Omron Sysmac Studio project servo_limites (Sysmac Studio 1.23.0.14, StandardProject)

# Controller new_Controller_0: NX1P2-1040DT1 version 1.18
Axis eje_1, settings changed from default: AxisType=ServoType, UnitsConversion=EnumElement2, UnitsNumerator=8380608, UnitsDenominator=143, MaxVelocity=50, MaxJogVelocity=20, HomingMode=BackupAndPressingTime, StartDirection=NegativeDirection, OriginInputDetectionDirection=NegativeDirection, HomingVelocity=3, HomingApproachVelocity=1, HomingAcceleration=4, PushTime=1000, OriginCompensationValue=10, CompensationVelocity=0.5, ModuloMAXPosition=360, ModuloMINPosition=0, EncoderTypes=Abs
Task PrimaryTask (priority 4, period or condition 2000): Programa0

VAR_GLOBAL CONSTANT
    eje_1 : _sAXIS_REF;  (* at MC://_MC_AX[0] *)
END_VAR

PROGRAM Programa0
VAR
    servo_on : BOOL;
    et10 : BOOL;
    on_servo : BOOL;
    et11 : BOOL;
    et12 : BOOL;
    reset_servo1 : MC_Reset;
    power_servo1 : MC_Power;
    home_servo : MC_Home;
    absolute1_servo1 : MC_MoveAbsolute;
    abs_move : BOOL;
    et0 : BOOL;
    et1 : BOOL;
    et2 : BOOL;
    eje1 : _sAXIS_REF;
END_VAR
VAR_EXTERNAL CONSTANT
    eje_1 : _sAXIS_REF;
END_VAR

(* Section activar: ladder, written here as Structured Text *)

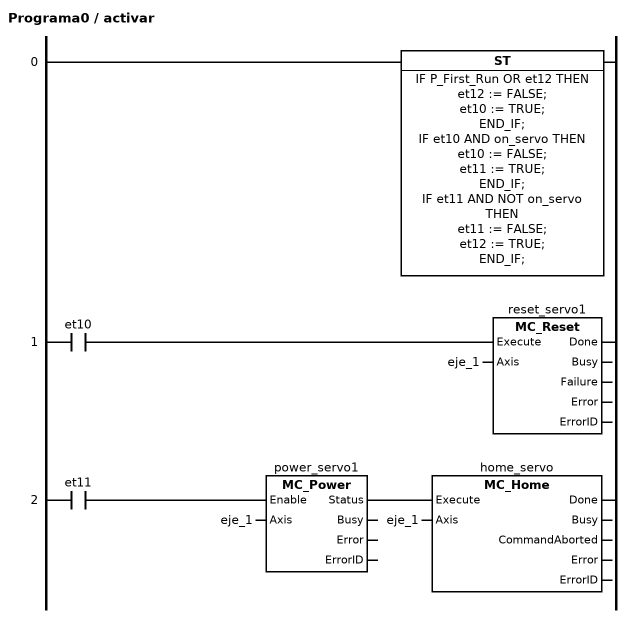
(* Rung 0 *)
IF P_First_Run OR et12 THEN
	et12 := FALSE;
	et10 := TRUE;
END_IF;
IF et10 AND on_servo THEN
	et10 := FALSE;
	et11 := TRUE;
END_IF;
IF et11 AND NOT on_servo THEN
	et11 := FALSE;
	et12 := TRUE;
END_IF;
(* Rung 1 *)
reset_servo1(Execute := et10, Axis := eje_1);
(* Rung 2 *)
power_servo1(Enable := et11, Axis := eje_1);
home_servo(Execute := power_servo1.Status, Axis := eje_1);

(* Section produccion: ladder, written here as Structured Text *)

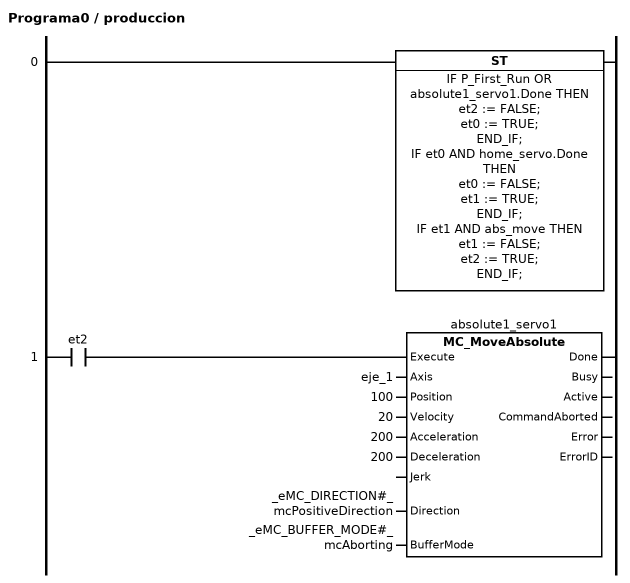
(* Rung 0 *)
IF P_First_Run OR absolute1_servo1.Done THEN
	et2 := FALSE;
	et0 := TRUE;
END_IF;
IF et0 AND home_servo.Done THEN
	et0 := FALSE;
	et1 := TRUE;
END_IF;
IF et1 AND abs_move THEN
	et1 := FALSE;
	et2 := TRUE;
END_IF;
(* Rung 1 *)
absolute1_servo1(Execute := et2, Axis := eje_1, Position := 100, Velocity := 20, Acceleration := 200, Deceleration := 200, Direction := _eMC_DIRECTION#_mcPositiveDirection, BufferMode := _eMC_BUFFER_MODE#_mcAborting);
END_PROGRAM